// Copyright (c) 2024 Loupe (https://loupe.team), provided under the MIT License.

INTERFACE IPLCopenConsumer EXTENDS __SYSTEM.IQueryInterface


METHOD Aborted : BOOL
VAR_INPUT
END_VAR
END_METHOD


PROPERTY Consume : BOOL
GET
END_GET
END_PROPERTY


METHOD Errored : BOOL
VAR_INPUT
  ID : INT;
END_VAR
END_METHOD


METHOD Finished : BOOL
VAR_INPUT
END_VAR
END_METHOD


PROPERTY Status : PLCopenStatusBase
GET
END_GET
END_PROPERTY

END_INTERFACE

(* stored: Version 1.1.0.1
   Itf IPLCopenConsumer: Id {6a7290ad-7ac6-41cc-ba9f-76967b5f2bc2}
   Method Aborted: Id {c13e0269-f6af-093a-3e84-237aad3bcb62}
   Property Consume: Id {6ba5532d-76e4-4a60-b32b-48609e504b06}
   Get Get: Id {fc1cb8fe-825b-4bd0-8ac5-01ed01104e14}
   Method Errored: Id {97e64f8a-ca69-4b1b-8dc4-ea125d2e68b1}
   Method Finished: Id {4dc5d1fd-a670-4a40-a328-0de89f694dac}
   Property Status: Id {9266aac4-62d7-464d-baa9-484a50b91022}
   Get Get: Id {96664bbd-85e9-4163-9d89-7e961369eeb2} *)
